// TIA Portal V16 export
// export: Created 2021-07-12T14:47:19.4175407Z, ExportSetting WithDefaults, DisplayName Totally Integrated Automation Portal, DisplayVersion V16, DisplayName TIA Portal Version Control Interface, DisplayVersion V16, DisplayName TIA Portal Openness, DisplayVersion V16, DisplayName STEP 7 Professional, DisplayVersion V16, DisplayName STEP 7 Safety, DisplayVersion V16, DisplayName WinCC Professional, DisplayVersion V16
TYPE "SimaHydTO_typeHMIConnectionBasicAxisControl"
TITLE = SimaHydTO_typeHMIConnectionBasicAxisControl
// HMI interface: Basic axis control (LAxisBasics)
// stored: IsFailsafeCompliant false
   STRUCT
      Command { S7_SetPoint := 'True'} : "SimaHydTO_typeHMIConnectionBasicAxisControlCommand";
      Status { S7_SetPoint := 'True'} : "SimaHydTO_typeHMIConnectionBasicAxisControlStatus";
      ControlDirectOutput { S7_SetPoint := 'True'} : "SimaHydTO_typeIHMIConnectionBasicAxisControlDirectOutput";
      StatusDirectOutput { S7_SetPoint := 'True'} : "SimaHydTO_typeHMIConnectionBasicAxislStatusDirectOutput";
   END_STRUCT;
END_TYPE
